// TIA Portal V17 export
// export: Created 2023-05-07T12:12:12.3788774Z, ExportSetting WithDefaults, DisplayName Totally Integrated Automation Portal, DisplayVersion V17, DisplayName TIA Portal Openness, DisplayVersion V17, DisplayName TIA Portal Version Control Interface, DisplayVersion V17, DisplayName TIA Portal Test Suite Advanced, DisplayVersion V17, DisplayName STEP 7 Professional, DisplayVersion V17, DisplayName SIMATIC Energy Suite, DisplayVersion V17, DisplayName STEP 7 Safety, DisplayVersion V17, DisplayName WinCC Professional, DisplayVersion V17
FUNCTION_BLOCK "RandomDisturbance"   // FB10, LAD
TITLE = RandomDisturbance
{ S7_Optimized_Access := 'TRUE' }
VERSION : 0.1
// stored: AutoNumber true, IsIECCheckEnabled false, IsRetainMemResEnabled false, MemoryReserve 100, SetENOAutomatically false, UDAEnableTagReadback false
   VAR_INPUT
      DistribanceMode : Int;
      Outflow : Int;
   END_VAR
   VAR_OUTPUT
      DischargeValve : Int;
   END_VAR
   VAR
      TON_1 { ExternalAccessible := 'False'; ExternalVisible := 'False'; ExternalWritable := 'False'} : TON_TIME;
      TON_2 { ExternalAccessible := 'False'; ExternalVisible := 'False'; ExternalWritable := 'False'} : TON_TIME;
      TP { ExternalAccessible := 'False'; ExternalVisible := 'False'; ExternalWritable := 'False'} : TP_TIME;
      TON_3 { ExternalAccessible := 'False'; ExternalVisible := 'False'; ExternalWritable := 'False'} : TON_TIME;
      random { S7_SetPoint := 'True'} : Int;
      p_Q : Bool;
   END_VAR
   VAR_TEMP   // added for the SCL form of the ladder/FBD networks
      _w1 : Bool;
   END_VAR
BEGIN

REGION Network 1: Disturbance
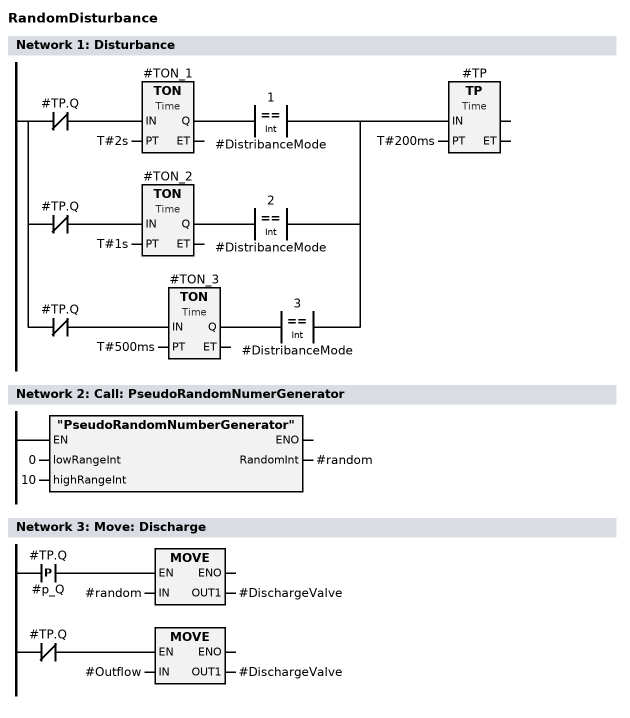
   RUNG wire#powerrail
      I_Contact( #TP.Q )
      { S7_Templates := "time_type := Time" } #TON_1.TON(pt := T#2s, et =>)
      { S7_Templates := "SrcType := Int" } EQ_Contact(in1 := 1, in2 := #DistribanceMode)
      wire#w1
      { S7_Templates := "time_type := Time" } #TP.TP(pt := T#200ms, et =>)
   END_RUNG
   RUNG wire#powerrail
      I_Contact( #TP.Q )
      { S7_Templates := "time_type := Time" } #TON_2.TON(pt := T#1s, et =>)
      { S7_Templates := "SrcType := Int" } EQ_Contact(in1 := 2, in2 := #DistribanceMode)
   END_RUNG wire#w1
   RUNG wire#powerrail
      I_Contact( #TP.Q )
      { S7_Templates := "time_type := Time" } #TON_3.TON(pt := T#500ms, et =>)
      { S7_Templates := "SrcType := Int" } EQ_Contact(in1 := 3, in2 := #DistribanceMode)
   END_RUNG wire#w1
   // the same network as SCL:
   #TON_1(IN := NOT #TP.Q, PT := T#2s);   // TON
   #TON_2(IN := NOT #TP.Q, PT := T#1s);   // TON
   #TON_3(IN := NOT #TP.Q, PT := T#500ms);   // TON
   #TP(IN := (#TON_1.Q AND (1 = #DistribanceMode)) OR (#TON_2.Q AND (2 = #DistribanceMode)) OR (#TON_3.Q AND (3 = #DistribanceMode)),   // TP
       PT := T#200ms);
END_REGION

REGION Network 2: Call: PseudoRandomNumerGenerator
   RUNG wire#powerrail
      "PseudoRandomNumberGenerator"(lowRangeInt := 0, highRangeInt := 10, RandomInt => #random)
   END_RUNG
   // the same network as SCL:
   "PseudoRandomNumberGenerator"(lowRangeInt := 0, highRangeInt := 10, RandomInt => #random);
END_REGION

REGION Network 3: Move: Discharge
   RUNG wire#powerrail
      P_Contact(operand := #TP.Q, bit := #p_Q)
      Move(in := #random, out1 => #DischargeValve)
   END_RUNG
   RUNG wire#powerrail
      I_Contact( #TP.Q )
      Move(in := #Outflow, out1 => #DischargeValve)
   END_RUNG
   // the same network as SCL:
   #_w1 := #TP.Q AND NOT #p_Q;   // rising edge of #TP.Q
   #p_Q := #TP.Q;
   IF #_w1 THEN #DischargeValve := #random; END_IF;
   IF NOT #TP.Q THEN #DischargeValve := #Outflow; END_IF;
END_REGION
END_FUNCTION_BLOCK
